(* PLC project Generated.project, CODESYS CODESYS V3.5 SP19 Patch 1 *)
(* stored: creationDateTime 2026-08-26T16:40:01.147385, modificationDateTime 2026-08-26T16:40:01.147385 *)

(* values of E_DiveSearchState: WAIT_PRECONDITIONS: Attente benne ouverte, positions et Kobold au repos; READY_TO_DESCEND: Prêt à assister une demande de descente; SEARCHING_IMMERSION: Descente : attente front 0->1 dans fenêtre eau; SEARCHING_BOTTOM: Immersion validée : attente front 1->0 au fond; BOTTOM_CONFIRMED: Fond validé ; extraction peut être demandée; ERROR_HOLD: Séquence invalide, descente assistée interdite *)

{attribute 'qualified_only'}
{attribute 'strict'}
TYPE E_DiveSearchState : (WAIT_PRECONDITIONS := 0, READY_TO_DESCEND := 1, SEARCHING_IMMERSION := 2, SEARCHING_BOTTOM := 3, BOTTOM_CONFIRMED := 4, ERROR_HOLD := 5);
END_TYPE
